TYPE Positive : ULINT; END_TYPE

(* stored: Version 1.1.0.1
   DUT Positive: Id {f81a29ed-500b-4d15-adb1-5fe8d87ec66d} *)
